// TIA Portal V19 export
DATA_BLOCK "SCALE AO_DB_2"   // DB149
// stored: InstanceOfName SCALE AO, InstanceOfType FB
"SCALE AO"
   // VAR_INPUT
   //    "SET RPM" : Real;
   //    "MIN RPM" : Real;
   //    "MAX RPM" : Real;
   //    "MIN RAW" : Int;
   //    "MAX RAW" : Int;
   // END_VAR
   // VAR_OUTPUT
   //    MODBUS : Int;
   // END_VAR
BEGIN
END_DATA_BLOCK
